Fanuc KAREL source: CA0051.KL

-- PROVISIONAL review KL for V770-1; original PC SHA256 7881d62658a8b6c853fd18e3079189034913a8886ed88ed750cb0b2c67c4264c
-- Incomplete behavior may be omitted. Consult companion uncertainty JSON. Do not deploy.
PROGRAM CA0051
%NOLOCKGROUP
BEGIN
  -- UNRESOLVED_PC offsets 0-1; opcodes 7B
  -- UNRESOLVED_PC offsets 6-20; opcodes 21,9D,52,23
  -- UNRESOLVED_PC offsets 25-29; opcodes 7F
  -- UNRESOLVED_PC offsets 34-41; opcodes 9C,23
  -- UNRESOLVED_PC offsets 46-53; opcodes 9D,23
  -- UNRESOLVED_PC offsets 58-69; opcodes 2E,23
  -- UNRESOLVED_PC offsets 74-81; opcodes 9D,23
  -- UNRESOLVED_PC offsets 86-95; opcodes 3F,75
  -- UNRESOLVED_PC offsets 100-114; opcodes 2E,22,9D,33,35
  -- UNRESOLVED_PC offsets 119-133; opcodes 2E,22,9D,33,35
  -- UNRESOLVED_PC offsets 138-153; opcodes 2E,22,32,35
  -- UNRESOLVED_PC offsets 158-173; opcodes 2E,22,32,35
  -- UNRESOLVED_PC offsets 178-410; opcodes 27,22,22,22,22,1C,22,22,22,22,22,1C,22,22,22,22,22,1C,22,22,22,22,22,1C,22,22,22,22,22,1C,22,22,22,22,22,1C,22,22,22,AA
  -- UNRESOLVED_PC offsets 415-419; opcodes 7F
END CA0051
